// TwinCAT 3 PLC project Untitled1
// ProgramVersion: 3.1.4023.0
// libraries:
//   Tc2_Standard, * (Beckhoff Automation GmbH)
//   Tc2_System, * (Beckhoff Automation GmbH)
//   TC3_EL6910_Backup_Restore, * (Beckhoff Automation GmbH)
//   Tc3_Module, * (Beckhoff Automation GmbH)
// project tree:
//   / PlcTask.TcTTO (not stored)
//   POUs/ FB_SafetyAutoLoad.TcPOU, MAIN.TcPOU, Safety_BckpRstr.TcPOU
// real-time tasks:
//   TASK PlcTask: cycle T#10ms, priority 20, ADS port 350
// motion (NC):
//   TASK NC-Task 1 SAF: cycle T#2ms, priority 4, ADS port 501
//   TASK NC-Task 1 SVB: cycle T#10ms, priority 8, ADS port 511
//   AXIS Axis 1 (id 1)
//     OtherSettings: AllowMotionCmdToSlave=true
//     encoder EncType=4
//       EncPara: MaxCount=#x0000ffff
//         Inc: RefSoftSyncMask=#x0000ffff
//     drive DrvType=24
//       Analog: TorqueSetpointScale=10, ScaleFactorActTorque=0.1
//       TimeComp: TaskDelayCycles=1
//     controller CtrType=1
//       CtrPara: PriorControlFactor=1
//         Observer: BandWidth=20
//   AXIS Axis 2 (id 2)
//     OtherSettings: AllowMotionCmdToSlave=true
//     encoder EncType=19
//       EncPara: MaxCount=#xffffffff
//     drive DrvType=16
//       DrvPara: MaxCount=#xffffffff, DriveControlDWord=#x00020000
//         Analog: TorqueSetpointScale=10, ScaleFactorActTorque=0.1
//         TimeComp: TaskDelayCycles=1
//     controller CtrType=1
//       CtrPara: PriorControlFactor=1
//         Observer: BandWidth=20
// I/O:
//   DEVICE Device 4 (EtherCAT), AmsNetId 172.18.232.94.5.1
//     Term 14 (EK1100) [EK1100 EtherCAT Coupler (2A E-Bus)]
//       Term 25 (EL2004) [EL2004 4Ch. Dig. Output 24V, 0.5A]
//       Term 26 (EL1018) [EL1018 8Ch. Dig. Input 24V, 10µs]
//       Term 27 (EL6900) [EL6900, TwinSAFE PLC]
//       Term 5 (EL9011) [EL9011 End Terminal]

// ---- POUs/FB_SafetyAutoLoad.TcPOU
FUNCTION_BLOCK FB_SafetyAutoLoad
VAR
	arEcNetId				AT %I* : T_AmsNetIdArr;
	nEcPort					AT %I* : WORD;
	arBufferBckpRstr		: ARRAY[0..16#FFFF] OF BYTE;
	sFileNameBckpRstr		: T_MaxString := 'C:\ProgramsToBeInstalled\Untitled2.bin';
	sNetIdRWFileBckpRstr	: T_AmsNetID := '5.25.217.162.1.1';	

	fbRestoreLogicProgram: FB_RESTORELOGICPROGRAM;
	refEcNetId: REFERENCE TO ARRAY [0..5] OF BYTE;
	refBuffer: REFERENCE TO ARRAY [0..16#FFFF] OF BYTE;
	nEcPort: WORD;
	sFileName: T_MaxString;
	sNetIdRWFile: T_AmsNetID;
END_VAR



fbRestoreLogicProgram(
	bExecute:= , 
	au8EcatNetId:= refEcNetId, 
	u16EcatPort:= nEcPort, 
	u32BufferAddress:= ADR(refBuffer), 
	u32BufferSize:= SIZEOF(refBuffer), 
	sFileName:= sFileName, 
	sNetIDReadFile:= sNetIdRWFile, );

END_FUNCTION_BLOCK

// ---- POUs/MAIN.TcPOU
PROGRAM MAIN
VAR
	Counter: INT;
	
	Safety_Reset AT %Q*:BOOL;
	Safety_Run AT %Q*:BOOL :=TRUE;
	Safety_ErroAck AT %Q*:BOOL;
END_VAR

Counter:=Counter+1;


Safety_BckpRstr();

END_PROGRAM

// ---- POUs/Safety_BckpRstr.TcPOU
PROGRAM Safety_BckpRstr
VAR
	/// Function to Get or Set device to specified state
	fbEcStateMachine: FB_EcStateMachine;
	stEcSlaveState: ST_EcSlaveState;
	stReqEcSlaveState: ST_EcSlaveState;
	stGetSlaveState: ST_TcGeneralOutputs;
	stSetSlaveState: ST_TcGeneralOutputs;
	/// better to be stored in File or on NOV-Ram
	nProjectSN: UDINT := 756788;
	/// better to be stored in File or on NOV-Ram
	nProjectCRC: WORD := 16#6207;
	/// Mapped to SerialNumber of EL69xx
	nFoundSN: UDINT;
	/// Mapped to CRC of EL69xx
	nFoundCRC: WORD;
	nStateCheckSn: UINT;
	bInit: BOOL := TRUE;
	bSnOk: BOOL;
	bCrcOk: BOOL;
	sMessageText: STRING;
	nTryCycle: INT;
	bErrAck: BOOL;
	/// #################################################
	/// CoE case functionality
	/// #################################################
	fbCoE_EL69xx: FB_CoE;
	iCoe: I_CoE;
	stCoE: ST_TcGeneralOutputs;
	ReadSafetyCoE: INT;
	bReadSafePlcInfoDone: BOOL;
	/// #############################################
	/// Backup and restore functionality
	/// #############################################
	fbSafetyBckpRstr: FB_SafetyAutoLoad;
	stSafetyBckpRstr: ST_TcOutputsSafetyBckpRstr;
	bRestore: BOOL;
	bBackup: BOOL;
	/// Visu-button to start restore
	bBtnRestore: BOOL;
	/// Visu-button to start backup
	bBtnBackup: BOOL;
	bProjectRestored: BOOL;
	bufEcNetId: ARRAY[0..5] OF BYTE;
	bReadSafePlcInfo: BOOL;
END_VAR

//##################################################
// Case condition of backup and restore
//##################################################
CASE nStateCheckSn OF
0: (* Init State *)
	sMessageText := '';
	//##################################################
	// Device state
	//##################################################
	fbEcStateMachine.NetId := F_CreateAmsNetId(nIds:= GVL_SafetyBckpRstr.arEcNetId); 
	fbEcStateMachine.SlaveAddr := WORD_TO_UINT(GVL_SafetyBckpRstr.nEcPort);
	fbEcStateMachine.ReqSlaveState(bExecute := FALSE);
	fbEcStateMachine.GetSlaveState(bExecute := FALSE);
	stReqEcSlaveState.deviceState := 0;
	nTryCycle := 0;
	//##################################################
	// Backup and restore
	//##################################################
	bRestore := FALSE;
	bBackup := FALSE;
	bReadSafePlcInfo := FALSE;
	fbSafetyBckpRstr.SaveLogicProgram(bExecute := FALSE);
	fbSafetyBckpRstr.RestoreLogicProgram(bExecute := FALSE);
	bufEcNetId := GVL_SafetyBckpRstr.arEcNetId;
	fbSafetyBckpRstr.EcNetId REF= bufEcNetId;
	fbSafetyBckpRstr.EcPort := GVL_SafetyBckpRstr.nEcPort;
	fbSafetyBckpRstr.Buffer REF= GVL_SafetyBckpRstr.arBufferBckpRstr;
	fbSafetyBckpRstr.NetIdRWFile := GVL_SafetyBckpRstr.sNetIdRWFileBckpRstr;
	fbSafetyBckpRstr.FileName := GVL_SafetyBckpRstr.sFileNameBckpRstr;
	
	IF bInit THEN
		stReqEcSlaveState.deviceState := EC_DEVICE_STATE_PREOP;
		nStateCheckSn := 20; // Get EL69xx
	END_IF
	//############################
	// Manual Backup
	IF bBtnBackup THEN
		nStateCheckSn := 100; // Backup safety project
	END_IF
	//############################
	// Manual Restore		
	IF bBtnRestore THEN
		nStateCheckSn := 110; // Restore safety project
	END_IF
		
10: (* Request State of EL69xx *)
	fbEcStateMachine.EcSetState := stReqEcSlaveState.deviceState;
	fbEcStateMachine.ReqSlaveState(bExecute := TRUE, stSetSlaveState => stSetSlaveState);
	
	IF NOT stSetSlaveState.bError THEN
		IF NOT stSetSlaveState.bBusy THEN
			fbEcStateMachine.ReqSlaveState(bExecute := FALSE);
			nStateCheckSn := 20;
		END_IF
	ELSE
		sMessageText := 'Error "Set State"';
		nStateCheckSn := 777;
	END_IF
	
20: (* GetSlaveState of EL69xx *)
	fbEcStateMachine.GetSlaveState(bExecute := TRUE, stGetSlaveState => stGetSlaveState);
	stEcSlaveState := fbEcStateMachine.EcGetState;
	
 	IF NOT stGetSlaveState.bError THEN
		IF NOT stGetSlaveState.bBusy AND (stEcSlaveState.deviceState = stReqEcSlaveState.deviceState) AND NOT bInit AND bRestore THEN
			fbEcStateMachine.GetSlaveState(bExecute := FALSE);
			nTryCycle := 0;
			nStateCheckSn := 110;
		ELSIF NOT stGetSlaveState.bBusy AND (stEcSlaveState.deviceState = stReqEcSlaveState.deviceState) AND NOT bInit THEN
			fbEcStateMachine.GetSlaveState(bExecute := FALSE);
			nTryCycle := 0;
			nStateCheckSn := 0;	
		ELSIF NOT stGetSlaveState.bBusy AND (stEcSlaveState.deviceState = stReqEcSlaveState.deviceState) AND bInit THEN
			fbEcStateMachine.GetSlaveState(bExecute := FALSE);
			nTryCycle := 0;
			nStateCheckSn := 30;
		ELSIF NOT stGetSlaveState.bBusy AND (stEcSlaveState.deviceState <> stReqEcSlaveState.deviceState) AND (nTryCycle < 9) THEN
			fbEcStateMachine.GetSlaveState(bExecute := FALSE);
			nTryCycle := nTryCycle + 1;
			nStateCheckSn := 10;
		ELSIF NOT stGetSlaveState.bBusy AND (stEcSlaveState.deviceState <> stReqEcSlaveState.deviceState) AND (nTryCycle >= 9) THEN
			fbEcStateMachine.GetSlaveState(bExecute := FALSE);
			nStateCheckSn := 777;
		END_IF
	ELSE
		sMessageText := 'Error "Get State"';
		nStateCheckSn := 777;
	END_IF
	
30: (* Check SN *)	
	bReadSafePlcInfo := TRUE; // Start CoE request of SafePlcInfoData
	IF bReadSafePlcInfoDone THEN
		IF (nProjectSN = nFoundSN) THEN
			bSnOk := TRUE;
			nStateCheckSn := 40; // Check CRC
		ELSE
			nProjectSN := nFoundSN;
			bSnOk := FALSE;
			nStateCheckSn := 40; // Check CRC
		END_IF	
	END_IF

40: (* Check CRC *)
	bInit := FALSE;
	IF (nProjectCRC = nFoundCRC) AND NOT  bProjectRestored THEN
		bCrcOk := TRUE;
		stReqEcSlaveState.deviceState := EC_DEVICE_STATE_OP;
		nStateCheckSn := 10; // Set EL69xx to OP
	ELSIF (nFoundCRC <> 0) AND bProjectRestored THEN
		nProjectCRC := nFoundCRC;
		bCrcOk := TRUE;
		nStateCheckSn := 0;
	ELSE 
		bCrcOk := FALSE;
		nStateCheckSn := 50; // Check CRC
	END_IF
	
50: (* CRC zero ? -> New EL69xx *)	
	IF (nFoundCRC = 0) THEN
		stReqEcSlaveState.deviceState := EC_DEVICE_STATE_OP;
		bRestore := TRUE;
		nStateCheckSn := 10; // Set EL69xx to OP		
	ELSE
		sMessageText := 'No way out! Download with engineering system!';
		nStateCheckSn := 777;	
	END_IF

100: (* Backup *)
	fbSafetyBckpRstr.SaveLogicProgram(bExecute := TRUE, stTcOutputsSafetyBckp => stSafetyBckpRstr);
	
	IF stSafetyBckpRstr.stTcGeneralOutputs.bError THEN
		sMessageText := 'Error "Backup"';
		nStateCheckSn := 777;
	ELSIF stSafetyBckpRstr.stTcGeneralOutputs.bDone  THEN
		nStateCheckSn := 0;
	END_IF
	
110: (* Restore Projekt *)
	fbSafetyBckpRstr.RestoreLogicProgram(bExecute := TRUE, stTcOutputsSafetyRstr => stSafetyBckpRstr);
	
	IF stSafetyBckpRstr.stTcGeneralOutputs.bError THEN
		sMessageText := 'Error "Restore"';
		nStateCheckSn := 777;
	ELSIF stSafetyBckpRstr.stTcGeneralOutputs.bDone  THEN
		bProjectRestored := TRUE;
		nStateCheckSn := 30; // Check SN and CRC again
	END_IF
777: (* Error *)
	IF bErrAck THEN
		sMessageText := '';
		stSafetyBckpRstr.sResult := '';
		nStateCheckSn := 0;
	END_IF
END_CASE

//##################################################
// Case condition of CoE read parameters of SafePLC
//##################################################
CASE ReadSafetyCoE OF
0: (* initialization *)	
	bReadSafePlcInfoDone := FALSE;
	IF bReadSafePlcInfo THEN
		bReadSafePlcInfo := FALSE;
		iCoE := fbCoE_EL69xx;
		iCoe.NetId := F_CreateAmsNetId(nIds:= GVL_SafetyBckpRstr.arEcNetId); 
		iCoE.SlaveAddress := 1008; // Address of EL69xx
		ReadSafetyCoE := 10;
	END_IF
	
10:	(* Read serial number of slave *)
	iCoE.Index := 16#F980;
	iCoE.SubIndex := 16#2;
	iCoE.DstBuf := ADR(nFoundSN);
	iCoE.BufLen := SIZEOF(nFoundSN);
	iCoE.CoERead(bExecute:=TRUE, stCoeRead=> stCoE);	
	
	IF stCoE.bError THEN
		ReadSafetyCoE := 777;
	ELSIF NOT stCoE.bBusy THEN
		iCoE.CoERead(bExecute:=FALSE, stCoeRead=> stCoE);
		ReadSafetyCoE := 30;
	END_IF

30:	(* Read crc of slave *)
	iCoE.Index := 16#F980;
	iCoE.SubIndex := 16#3;
	iCoE.DstBuf := ADR(nFoundCRC);
	iCoE.BufLen := SIZEOF(nFoundCRC);
	iCoE.CoERead(bExecute:=TRUE, stCoeRead=> stCoE);	
	
	IF stCoE.bError THEN
		ReadSafetyCoE := 777;
	ELSIF NOT stCoE.bBusy THEN
		iCoE.CoERead(bExecute:=FALSE, stCoeRead=> stCoE);
		bReadSafePlcInfoDone := TRUE;
		ReadSafetyCoE := 0;
	END_IF
	
777: (* Error *)
	IF bErrAck THEN
		ReadSafetyCoE := 0;
	END_IF
END_CASE

END_PROGRAM
